(* IEC 61131-3 sources: test/Class/_Radio32Ram, 1 file *)

(* ---- _Radio32Ram.st ---- *)
(*!
<Class
	Name               = "_Radio32Ram"
	Revision           = "0.1"
	RealtimeTask       = "false"
	CyclicTask         = "false"
	BackgroundTask     = "false"
	Sigmatek           = "true"
	OSInterface        = "false"
	HighPriority       = "false"
	Automatic          = "false"
	UpdateMode         = "Prescan"
	SharedCommandTable = "true"
	Objectsize         = "(284,120)"
	Comment            = "enables bitwise acces to 4 remanent Bytes, just one bit can be set to 1 all others are 0">
	<Channels>
		<Server Name="Data" Visualized="true" Initialize="false" WriteProtected="false" Retentive="false"/>
		<Client Name="RamData" Required="true" Internal="true"/>
	</Channels>
	<RevDoku>
		<Owner Company="sigmatek" Author="kolott"/>
		<Dokumentation Revision="0.1" Date="2011-09-28" Author="kolott" Company="sigmatek" Description="betterment datatypeconversion"/>
	</RevDoku>
	<Network Name="_Radio32Ram">
		<!-- List of Components in this network -->
		<Components>
			<Object
				Name       = "RamData"
				Class      = "Ram"
				Position   = "(0,0)"
				Visualized = "false">
				<Channels>
					<Server Name="Data"/>
				</Channels>
			</Object>
		</Components>
		<Comments>
		</Comments>
		<!-- List of Connections in this network -->
		<Connections>
			<Connection Source="this.RamData" Destination="RamData.Data"/>
		</Connections>
		<!-- Headerfiles -->
		<Options>
		</Options>
	</Network>
</Class>
*)
_Radio32Ram : CLASS
  //Servers:
	Data 	: SvrChCmd_BDINT;
  //Clients:
	RamData 	: CltChCmd_Ram;
  //Variables:
  //Functions:

	FUNCTION VIRTUAL GLOBAL Data::Read
		VAR_OUTPUT
			output (EAX) 	: BDINT;
		END_VAR;

	FUNCTION VIRTUAL GLOBAL Data::Write
		VAR_INPUT
			input (EAX) 	: BDINT;
		END_VAR
		VAR_OUTPUT
			result (EAX) 	: BDINT;
		END_VAR;
  //Tables:
	FUNCTION @STD
		VAR_OUTPUT
			ret_code	: CONFSTATES;
		END_VAR;
	FUNCTION GLOBAL TAB @CT_;
END_CLASS;

#pragma using Ram

//*********************Inserted from .\_Radio32Ram\_Radio32Ram_00_00.st*********************

FUNCTION VIRTUAL GLOBAL _Radio32Ram::Data::Read
	VAR_OUTPUT
		output (EAX) 	: BDINT;
	END_VAR

  output$dint := RamData.Data.Read();

END_FUNCTION //VIRTUAL GLOBAL _Radio32Ram::Data::Read

FUNCTION VIRTUAL GLOBAL _Radio32Ram::Data::Write
	VAR_INPUT
		input (EAX) 	: BDINT;
	END_VAR
	VAR_OUTPUT
		result (EAX) 	: BDINT;
	END_VAR
VAR
    mydat : UDINT;
	para  : UDINT;
END_VAR

  mydat$DINT := RamData.Data.Read();
  para       := input$UDINT;

  if(para and 16#80000000) then
    if(para = 16#80000000) then
	  mydat := 16#80000000;
	else
      mydat := para and 16#7FFFFFFF;
    end_if;
  else
    if(para = 0) then
      mydat := mydat and 16#7FFFFFFF;
    else
	  mydat := mydat and (16#FFFFFFFF xor para);
	end_if;
  end_if;

  result:= mydat;
  Data  := mydat;
  RamData.Data.Write(result$dint);

END_FUNCTION //VIRTUAL GLOBAL _Radio32Ram::Data::Write
